Yaskawa INFORM job: kufsa_with_table_real.JBI

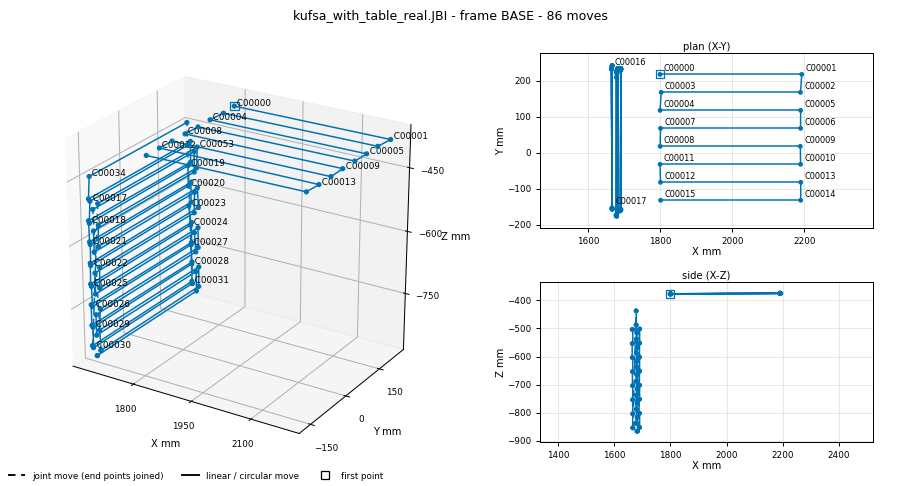
[picture p0: tool path of kufsa_with_table_real.JBI in frame BASE, 86 of 91 moves have a stored position in this frame; points joined in program order, loops and branches not executed]
/JOB
//NAME kufsa_with_table_real
//POS
///NPOS 86,0,86,0,0,0
///TOOL 0
///POSTYPE BASE
///RECTAN
///RCONF 1,0,0,0,0,0,0,0,0,0,0,0,0,0,0,0,0,0,0,0,0,0,0,0
C00000=1799.105440,217.743638,-376.719388,180.000000,0.000000,0.000000
C00001=2193.209433,217.743638,-375.224026,180.000000,0.000000,0.000000
C00002=2189.640761,167.743638,-375.035908,180.000000,0.000000,0.000000
C00003=1802.416487,167.743638,-376.945674,180.000000,0.000000,0.000000
C00004=1799.461545,117.743638,-377.155681,180.000000,0.000000,0.000000
C00005=2190.175047,117.743638,-375.229868,180.000000,0.000000,0.000000
C00006=2189.945342,67.743638,-374.707578,180.000000,0.000000,0.000000
C00007=1800.555244,67.743638,-377.416008,180.000000,0.000000,0.000000
C00008=1799.574494,17.743638,-377.432600,180.000000,0.000000,0.000000
C00009=2189.258004,17.743638,-374.777918,180.000000,0.000000,0.000000
C00010=2189.936458,-32.256362,-375.068157,180.000000,0.000000,0.000000
C00011=1799.279812,-32.256362,-377.528411,180.000000,0.000000,0.000000
C00012=1800.458286,-82.256362,-376.642738,180.000000,0.000000,0.000000
C00013=2190.469729,-82.256362,-375.087553,180.000000,0.000000,0.000000
C00014=2190.131390,-132.256362,-373.628646,180.000000,0.000000,0.000000
C00015=1800.792310,-132.256362,-376.594833,180.000000,0.000000,0.000000
C00016=1663.630321,232.602754,-503.508351,180.000000,-89.999999,0.000000
C00017=1666.148443,-152.983175,-503.508351,180.000000,-89.999999,0.000000
C00018=1666.041586,-157.222392,-553.508351,180.000000,-89.999999,0.000000
C00019=1663.921957,233.381709,-553.508351,180.000000,-89.999999,0.000000
C00020=1664.032114,233.772267,-603.508351,180.000000,-89.999999,0.000000
C00021=1666.195146,-156.635353,-603.508351,180.000000,-89.999999,0.000000
C00022=1666.144382,-156.750888,-653.508351,180.000000,-89.999999,0.000000
C00023=1664.648636,233.958899,-653.508351,180.000000,-89.999999,0.000000
C00024=1665.281911,240.186938,-703.508351,180.000000,-89.999999,0.000000
C00025=1666.323069,-156.758574,-703.508351,180.000000,-89.999999,0.000000
C00026=1665.536997,-154.099606,-753.508351,180.000000,-89.999999,0.000000
C00027=1665.709339,240.892633,-753.508351,180.000000,-89.999999,0.000000
C00028=1665.769494,242.378004,-803.508351,180.000000,-89.999999,0.000000
C00029=1665.928891,-154.891772,-803.508351,180.000000,-89.999999,0.000000
C00030=1665.831933,-155.041414,-853.508351,180.000000,-89.999999,0.000000
C00031=1666.587801,242.208666,-853.508351,180.000000,-89.999999,0.000000
C00032=1666.587801,242.208666,-853.508351,180.000000,-89.999999,0.000000
C00033=1677.678127,209.846616,-437.485725,180.000000,-89.999999,0.000000
C00034=1678.733788,-170.147797,-437.485725,180.000000,-89.999999,0.000000
C00035=1678.640352,-174.851541,-487.485725,180.000000,-89.999999,0.000000
C00036=1677.720161,223.186368,-487.485725,180.000000,-89.999999,0.000000
C00037=1679.116660,221.336801,-537.485725,180.000000,-89.999999,0.000000
C00038=1678.510406,-176.882587,-537.485725,180.000000,-89.999999,0.000000
C00039=1678.539950,-175.322372,-587.485725,180.000000,-89.999999,0.000000
C00040=1678.922822,222.387098,-587.485725,180.000000,-89.999999,0.000000
C00041=1677.674044,223.803652,-637.485725,180.000000,-89.999999,0.000000
C00042=1678.841396,-175.651065,-637.485725,180.000000,-89.999999,0.000000
C00043=1678.086460,-175.495729,-687.485725,180.000000,-89.999999,0.000000
C00044=1678.879827,222.804373,-687.485725,180.000000,-89.999999,0.000000
C00045=1679.569189,221.289337,-737.485725,180.000000,-89.999999,0.000000
C00046=1677.443696,-175.016268,-737.485725,180.000000,-89.999999,0.000000
C00047=1677.458828,-174.730216,-787.485725,180.000000,-89.999999,0.000000
C00048=1679.429395,222.793205,-787.485725,180.000000,-89.999999,0.000000
C00049=1678.605764,222.672896,-837.485725,180.000000,-89.999999,0.000000
C00050=1677.393735,-173.939575,-837.485725,180.000000,-89.999999,0.000000
C00051=1677.393735,-173.939575,-837.485725,180.000000,-89.999999,0.000000
C00052=1690.476739,-158.083429,-501.808827,180.000000,-89.999999,0.000000
C00053=1690.334602,232.310020,-501.808827,180.000000,-89.999999,0.000000
C00054=1690.515066,228.872097,-551.808827,180.000000,-89.999999,0.000000
C00055=1690.213912,-157.792792,-551.808827,180.000000,-89.999999,0.000000
C00056=1689.886360,-159.444379,-601.808827,180.000000,-89.999999,0.000000
C00057=1690.200332,231.911776,-601.808827,180.000000,-89.999999,0.000000
C00058=1690.555169,234.541680,-651.808827,180.000000,-89.999999,0.000000
C00059=1690.322418,-157.870855,-651.808827,180.000000,-89.999999,0.000000
C00060=1689.273645,-157.628738,-701.808827,180.000000,-89.999999,0.000000
C00061=1690.491461,232.591770,-701.808827,180.000000,-89.999999,0.000000
C00062=1690.566845,232.330677,-751.808827,180.000000,-89.999999,0.000000
C00063=1689.218059,-157.905924,-751.808827,180.000000,-89.999999,0.000000
C00064=1688.411428,-162.050263,-801.808827,180.000000,-89.999999,0.000000
C00065=1690.582835,234.258249,-801.808827,180.000000,-89.999999,0.000000
C00066=1690.493999,233.192980,-851.808827,180.000000,-89.999999,0.000000
C00067=1689.187855,-159.833976,-851.808827,180.000000,-89.999999,0.000000
C00068=1689.187855,-159.833976,-851.808827,180.000000,-89.999999,0.000000
C00069=1680.766998,-163.387450,-515.527796,180.000000,-89.999999,0.000000
C00070=1680.834974,234.142317,-515.527796,180.000000,-89.999999,0.000000
C00071=1680.687013,233.311065,-565.527796,180.000000,-89.999999,0.000000
C00072=1681.066523,-163.618677,-565.527796,180.000000,-89.999999,0.000000
C00073=1681.334101,-163.573244,-615.527796,180.000000,-89.999999,0.000000
C00074=1681.446272,233.261063,-615.527796,180.000000,-89.999999,0.000000
C00075=1681.738110,230.395973,-665.527796,180.000000,-89.999999,0.000000
C00076=1681.212562,-162.975504,-665.527796,180.000000,-89.999999,0.000000
C00077=1681.395831,-163.194802,-715.527796,180.000000,-89.999999,0.000000
C00078=1681.907689,230.406887,-715.527796,180.000000,-89.999999,0.000000
C00079=1682.792090,233.976828,-765.527796,180.000000,-89.999999,0.000000
C00080=1681.078773,-163.308512,-765.527796,180.000000,-89.999999,0.000000
C00081=1681.118885,-163.048857,-815.527796,180.000000,-89.999999,0.000000
C00082=1683.164874,233.406500,-815.527796,180.000000,-89.999999,0.000000
C00083=1683.638300,234.090284,-865.527796,180.000000,-89.999999,0.000000
C00084=1681.192626,-162.997079,-865.527796,180.000000,-89.999999,0.000000
C00085=1681.192626,-162.997079,-865.527796,180.000000,-89.999999,0.000000
///POSTYPE PULSE
///PULSE
EC00000=0
EC00001=0
EC00002=0
EC00003=0
EC00004=0
EC00005=0
EC00006=0
EC00007=0
EC00008=0
EC00009=0
EC00010=0
EC00011=0
EC00012=0
EC00013=0
EC00014=0
EC00015=0
EC00016=0
EC00017=0
EC00018=0
EC00019=0
EC00020=0
EC00021=0
EC00022=0
EC00023=0
EC00024=0
EC00025=0
EC00026=0
EC00027=0
EC00028=0
EC00029=0
EC00030=0
EC00031=0
EC00032=92160
EC00033=92160
EC00034=92160
EC00035=92160
EC00036=92160
EC00037=92160
EC00038=92160
EC00039=92160
EC00040=92160
EC00041=92160
EC00042=92160
EC00043=92160
EC00044=92160
EC00045=92160
EC00046=92160
EC00047=92160
EC00048=92160
EC00049=92160
EC00050=92160
EC00051=184320
EC00052=184320
EC00053=184320
EC00054=184320
EC00055=184320
EC00056=184320
EC00057=184320
EC00058=184320
EC00059=184320
EC00060=184320
EC00061=184320
EC00062=184320
EC00063=184320
EC00064=184320
EC00065=184320
EC00066=184320
EC00067=184320
EC00068=276480
EC00069=276480
EC00070=276480
EC00071=276480
EC00072=276480
EC00073=276480
EC00074=276480
EC00075=276480
EC00076=276480
EC00077=276480
EC00078=276480
EC00079=276480
EC00080=276480
EC00081=276480
EC00082=276480
EC00083=276480
EC00084=276480
EC00085=368640
//INST
///DATE 2023/01/17 15:13
///ATTR SC,RW,RJ
////FRAME BASE
///GROUP1 RB1,ST1
NOP
MOVJ C00000 EC00000 VJ=15.0
CALL JOB:SPYON
MOVL C00001 EC00001 V=200.0
MOVL C00002 EC00002 V=200.0
MOVL C00003 EC00003 V=200.0
MOVL C00004 EC00004 V=200.0
MOVL C00005 EC00005 V=200.0
MOVL C00006 EC00006 V=200.0
MOVL C00007 EC00007 V=200.0
MOVL C00008 EC00008 V=200.0
MOVL C00009 EC00009 V=200.0
MOVL C00010 EC00010 V=200.0
MOVL C00011 EC00011 V=200.0
MOVL C00012 EC00012 V=200.0
MOVL C00013 EC00013 V=200.0
MOVL C00014 EC00014 V=200.0
MOVL C00015 EC00015 V=200.0
CALL JOB:SPYOF
MOVJ P009 VJ=15.00
MOVJ C00016 EC00016 VJ=15.0
CALL JOB:SPYON
MOVL C00017 EC00017 V=200.0
MOVL C00018 EC00018 V=200.0
MOVL C00019 EC00019 V=200.0
MOVL C00020 EC00020 V=200.0
MOVL C00021 EC00021 V=200.0
MOVL C00022 EC00022 V=200.0
MOVL C00023 EC00023 V=200.0
MOVL C00024 EC00024 V=200.0
MOVL C00025 EC00025 V=200.0
MOVL C00026 EC00026 V=200.0
MOVL C00027 EC00027 V=200.0
MOVL C00028 EC00028 V=200.0
MOVL C00029 EC00029 V=200.0
MOVL C00030 EC00030 V=200.0
MOVL C00031 EC00031 V=200.0
CALL JOB:SPYOF
MOVJ P009 VJ=15.00
MOVL C00032 EC00032 V=200.0
MOVJ C00033 EC00033 VJ=15.0
CALL JOB:SPYON
MOVL C00034 EC00034 V=200.0
MOVL C00035 EC00035 V=200.0
MOVL C00036 EC00036 V=200.0
MOVL C00037 EC00037 V=200.0
MOVL C00038 EC00038 V=200.0
MOVL C00039 EC00039 V=200.0
MOVL C00040 EC00040 V=200.0
MOVL C00041 EC00041 V=200.0
MOVL C00042 EC00042 V=200.0
MOVL C00043 EC00043 V=200.0
MOVL C00044 EC00044 V=200.0
MOVL C00045 EC00045 V=200.0
MOVL C00046 EC00046 V=200.0
MOVL C00047 EC00047 V=200.0
MOVL C00048 EC00048 V=200.0
MOVL C00049 EC00049 V=200.0
MOVL C00050 EC00050 V=200.0
CALL JOB:SPYOF
MOVJ P009 VJ=15.00
MOVL C00051 EC00051 V=200.0
MOVJ C00052 EC00052 VJ=15.0
CALL JOB:SPYON
MOVL C00053 EC00053 V=200.0
MOVL C00054 EC00054 V=200.0
MOVL C00055 EC00055 V=200.0
MOVL C00056 EC00056 V=200.0
MOVL C00057 EC00057 V=200.0
MOVL C00058 EC00058 V=200.0
MOVL C00059 EC00059 V=200.0
MOVL C00060 EC00060 V=200.0
MOVL C00061 EC00061 V=200.0
MOVL C00062 EC00062 V=200.0
MOVL C00063 EC00063 V=200.0
MOVL C00064 EC00064 V=200.0
MOVL C00065 EC00065 V=200.0
MOVL C00066 EC00066 V=200.0
MOVL C00067 EC00067 V=200.0
CALL JOB:SPYOF
MOVJ P009 VJ=15.00
MOVL C00068 EC00068 V=200.0
MOVJ C00069 EC00069 VJ=15.0
CALL JOB:SPYON
MOVL C00070 EC00070 V=200.0
MOVL C00071 EC00071 V=200.0
MOVL C00072 EC00072 V=200.0
MOVL C00073 EC00073 V=200.0
MOVL C00074 EC00074 V=200.0
MOVL C00075 EC00075 V=200.0
MOVL C00076 EC00076 V=200.0
MOVL C00077 EC00077 V=200.0
MOVL C00078 EC00078 V=200.0
MOVL C00079 EC00079 V=200.0
MOVL C00080 EC00080 V=200.0
MOVL C00081 EC00081 V=200.0
MOVL C00082 EC00082 V=200.0
MOVL C00083 EC00083 V=200.0
MOVL C00084 EC00084 V=200.0
CALL JOB:SPYOF
MOVJ P009 VJ=15.00
MOVL C00085 EC00085 V=200.0
END
